FUNCTION fun_AreaM_SPEGNITUTTO : FB_Semaforo
VAR_INPUT
END_VAR
VAR
	bT3EnTPausaLavoro: BOOL;
END_VAR


//bit di COMANDO (cmd nellinterfaccia)
bT1_ON:=FALSE;
bT2_ON:=FALSE;
bT3_ON:=FALSE;
T3_ModoPausaLavoro:=FALSE;
bT3EnT1PausaLavoro:=FALSE;
bT3EnT2PausaLavoro:=FALSE;
T3_Lavoro :=FALSE;	
M_Start_Macinatore_Loc := FALSE;
bT4_ON:=FALSE;
bM_ON:=FALSE;


bMacinatoreStop:=TRUE;
bMacinatoreStart:=FALSE;
bT3T5T6DelayStart:=FALSE;

//uscite finali
HQ1_T1_KA1:=FALSE;
HQ1_T2_KA2:=FALSE;
HQ1_T3_KA3:=FALSE;
HQ1_T4_KA4:=FALSE;
HQ1_T5_KA5:=FALSE;
HQ1_T6_KA6:=FALSE;

//macchine a stati
stepT1T2:=100;
stepT3:=100;
stepT4:=100;
descT1T2:='T1-T2 disabilitati';
descT3:='T3 disabilitati';
descT4:='T4 disabilitati';

END_FUNCTION

(* stored: Version 1.1.0.1, ProductVersion 3.1.4022.12
   POU fun_AreaM_SPEGNITUTTO: Id {35fdccf8-d760-4663-b4ef-f1804d1ac664}, SpecialFunc None *)
